// TwinCAT 3 PLC project Motion
// ProgramVersion: 3.1.4022.0
// libraries:
//   Tc2_MC2, * (Beckhoff Automation GmbH)
//   Tc2_Standard, * (Beckhoff Automation GmbH)
//   Tc2_System, * (Beckhoff Automation GmbH)
//   Tc3_Module, * (Beckhoff Automation GmbH)
//   VisuSymbols,3.5.10.0,System
// project tree:
//   / GlobalTextList.TcGTLO (not stored), PlcTask.TcTTO, VisualizationManager.TcVMO (not stored), VISU_TASK.TcTTO (not stored)
//   GVLs/ GVL_ver.TcGVL
//   POUs/ Axis2.TcPOU, Axis3.TcPOU (not stored), Axis4.TcPOU, Axis5.TcPOU (not stored), Axis6.TcPOU (not stored), Axis7.TcPOU (not stored), Axis8.TcPOU, Axis9.TcPOU (not stored), Axis10.TcPOU, GCC2.TcPOU (not stored), LadderLogic.TcPOU, MAIN.TcPOU, Axis1.TcPOU (not stored), GCC1.TcPOU
//   VISUs/ StandMotors.TcVIS, ManiMotors.TcVIS
// real-time tasks:
//   TASK PlcTask: cycle T#10ms, priority 20, ADS port 350
//   TASK VISU_TASK: cycle T#200000us, priority 30, ADS port 351
// motion (NC):
//   TASK NC-Task 1 SAF: cycle T#2ms, priority 4, ADS port 501
//   TASK NC-Task 1 SVB: cycle T#10ms, priority 8, ADS port 511
//   AXIS Axis 2 (id 2)
//     Dynamic: Acceleration=4, Deceleration=4, Jerk=4, AccelerationMaximum=4, DecelerationMaximum=4
//     Velo: RefSearch=0.3125, RefSync=0.3125, SlowManual=0.15625, FastManual=0.3125, Maximum=1
//     BacklashCompensation: Enable=true
//     OtherSettings: AllowMotionCmdToSlave=true, PulseDistancePos=0.015625, PulseDistanceNeg=0.015625
//     encoder EncType=4
//       EncPara: ScaleFactorNumerator=0.00015625, MaxCount=#x0000ffff
//         ActPosCorrection: Enable=true, Time=0.02
//         Inc: RefSoftSyncMask=#x0000ffff
//     drive DrvType=24
//       Analog: VeloReferenz=2, ScaleFactorActTorque=0.1
//       TimeComp: TaskDelayCycles=1
//     controller CtrType=1
//       CtrPara: PriorControlFactor=1
//         Observer: BandWidth=20
//   AXIS Axis 3 (id 3)
//     Dynamic: Acceleration=4, Deceleration=4, Jerk=4, AccelerationMaximum=4, DecelerationMaximum=4
//     Velo: RefSearch=0.3125, RefSync=0.3125, SlowManual=0.015625, FastManual=0.3125, Maximum=1
//     BacklashCompensation: Enable=true
//     OtherSettings: AllowMotionCmdToSlave=true, PulseDistancePos=0.015625
//     encoder EncType=4
//       EncPara: ScaleFactorNumerator=7.8125e-06, MaxCount=#x0000ffff
//         ActPosCorrection: Enable=true, Time=0.02
//         Inc: RefSoftSyncMask=#x0000ffff
//     drive DrvType=24
//       Analog: VeloReferenz=2, ScaleFactorActTorque=0.1
//       TimeComp: TaskDelayCycles=1
//     controller CtrType=1
//       CtrPara: PriorControlFactor=1
//         Observer: BandWidth=20
//   AXIS Axis 4 (id 4)
//     Dynamic: Acceleration=4, Deceleration=4, Jerk=4, AccelerationMaximum=4, DecelerationMaximum=4
//     Velo: RefSearch=0.3125, RefSync=0.3125, SlowManual=0.15625, FastManual=0.3125, Maximum=1
//     BacklashCompensation: Enable=true
//     OtherSettings: PulseDistancePos=0.015625, PulseDistanceNeg=0.015625
//     encoder EncType=4
//       EncPara: ScaleFactorNumerator=0.00015625, MaxCount=#x0000ffff
//         SoftEndMinControl: Enable=true, Range=-2.1
//         SoftEndMaxControl: Enable=true, Range=6.1
//         ActPosCorrection: Enable=true, Time=0.02
//         Inc: RefSoftSyncMask=#x0000ffff
//     drive DrvType=24
//       Analog: VeloReferenz=2, ScaleFactorActTorque=0.1
//       TimeComp: TaskDelayCycles=1
//     controller CtrType=1
//       CtrPara: PriorControlFactor=1
//         PosDiffControl: Range=1
//         Observer: BandWidth=20
//   AXIS Axis 5 (id 5)
//     Dynamic: Acceleration=4, Deceleration=4, Jerk=4, AccelerationMaximum=4, DecelerationMaximum=4
//     Velo: RefSearch=0.3125, RefSync=0.3125, SlowManual=0.15625, FastManual=0.3125, Maximum=1
//     BacklashCompensation: Enable=true
//     OtherSettings: AllowMotionCmdToSlave=true, PulseDistancePos=0.015625, PulseDistanceNeg=0.015625
//     encoder EncType=4
//       EncPara: ScaleFactorNumerator=7.8125e-06, MaxCount=#x0000ffff
//         ActPosCorrection: Enable=true, Time=0.02
//         Inc: RefSoftSyncMask=#x0000ffff
//     drive DrvType=24
//       Analog: VeloReferenz=2, ScaleFactorActTorque=0.1
//       TimeComp: TaskDelayCycles=1
//     controller CtrType=1
//       CtrPara: PriorControlFactor=1
//         Observer: BandWidth=20
//   AXIS Axis 6 (id 6)
//     Dynamic: Acceleration=4, Deceleration=4, Jerk=4, AccelerationMaximum=4, DecelerationMaximum=4
//     Velo: RefSearch=0.3125, RefSync=0.3125, SlowManual=0.15625, FastManual=0.3125, Maximum=1
//     BacklashCompensation: Enable=true
//     OtherSettings: AllowMotionCmdToSlave=true, PulseDistancePos=0.015625, PulseDistanceNeg=0.015625
//     encoder EncType=4
//       EncPara: ScaleFactorNumerator=0.00015625, MaxCount=#x0000ffff
//         ActPosCorrection: Enable=true, Time=0.02
//         Inc: RefSoftSyncMask=#x0000ffff
//     drive DrvType=24
//       Analog: VeloReferenz=2, ScaleFactorActTorque=0.1
//       TimeComp: TaskDelayCycles=1
//     controller CtrType=1
//       CtrPara: PriorControlFactor=1
//         Observer: BandWidth=20
//   AXIS Axis 7 (id 7)
//     Dynamic: Acceleration=4, Deceleration=4, Jerk=4, AccelerationMaximum=4, DecelerationMaximum=4
//     Velo: RefSearch=0.3125, RefSync=0.3125, SlowManual=0.15625, FastManual=0.3125, Maximum=1
//     BacklashCompensation: Enable=true
//     OtherSettings: AllowMotionCmdToSlave=true, PulseDistancePos=0.015625, PulseDistanceNeg=0.015625
//     encoder EncType=1
//       EncPara: ScaleFactorNumerator=1.5625e-05
//         ActPosCorrection: Enable=true, Time=0.02
//         Inc: RefSoftSyncMask=#x0000ffff
//     drive DrvType=24
//       Analog: VeloReferenz=2, ScaleFactorActTorque=0.1
//       TimeComp: TaskDelayCycles=1
//     controller CtrType=1
//       CtrPara: PriorControlFactor=1
//         Observer: BandWidth=20
//   AXIS Axis 8 (id 8)
//     Dynamic: Acceleration=4, Deceleration=4, Jerk=4, AccelerationMaximum=4, DecelerationMaximum=4
//     Velo: RefSearch=0.3125, RefSync=0.3125, SlowManual=0.15625, FastManual=0.3125, Maximum=1
//     BacklashCompensation: Enable=true
//     OtherSettings: AllowMotionCmdToSlave=true, PulseDistancePos=0.015625, PulseDistanceNeg=0.015625
//     encoder EncType=4
//       EncPara: ScaleFactorNumerator=1.5625e-05, MaxCount=#x0000ffff
//         ActPosCorrection: Enable=true, Time=0.02
//         Inc: RefSoftSyncMask=#x0000ffff
//     drive DrvType=24
//       Analog: VeloReferenz=2, ScaleFactorActTorque=0.1
//       TimeComp: TaskDelayCycles=1
//     controller CtrType=1
//       CtrPara: PriorControlFactor=1
//         Observer: BandWidth=20
//   AXIS Axis 9 (id 9)
//     Dynamic: Acceleration=4, Deceleration=4, Jerk=4, AccelerationMaximum=4, DecelerationMaximum=4
//     Velo: RefSearch=0.3125, RefSync=0.3125, SlowManual=0.15625, FastManual=0.3125, Maximum=1
//     BacklashCompensation: Enable=true
//     OtherSettings: AllowMotionCmdToSlave=true, PulseDistancePos=0.015625, PulseDistanceNeg=0.015625
//     encoder EncType=4
//       EncPara: ScaleFactorNumerator=7.812e-05, MaxCount=#x0000ffff
//         ActPosCorrection: Enable=true, Time=0.02
//         Inc: RefSoftSyncMask=#x0000ffff
//     drive DrvType=24
//       Analog: VeloReferenz=2, ScaleFactorActTorque=0.1
//       TimeComp: TaskDelayCycles=1
//     controller CtrType=1
//       CtrPara: PriorControlFactor=1
//         Observer: BandWidth=20
//   AXIS Axis 10 (id 10)
//     General: UnitName=°
//     Dynamic: Acceleration=4, Deceleration=4, Jerk=4, AccelerationMaximum=4, DecelerationMaximum=4
//     Velo: RefSearch=0.3125, RefSync=0.3125, SlowManual=0.15625, FastManual=0.3125, Maximum=1
//     BacklashCompensation: Enable=true
//     OtherSettings: AllowMotionCmdToSlave=true, PulseDistancePos=0.015625, PulseDistanceNeg=0.015625
//     encoder EncType=4
//       EncPara: ScaleFactorNumerator=0.00028125, MaxCount=#x0000ffff
//         ActPosCorrection: Enable=true, Time=0.02
//         Inc: RefSoftSyncMask=#x0000ffff
//     drive DrvType=24
//       Analog: VeloReferenz=2, ScaleFactorActTorque=0.1
//       TimeComp: TaskDelayCycles=1
//     controller CtrType=1
//       CtrPara: PriorControlFactor=1
//         Observer: BandWidth=20
//   AXIS Axis 1 (id 1)
//     Dynamic: Acceleration=4, Deceleration=4, Jerk=4, AccelerationMaximum=4, DecelerationMaximum=4
//     Velo: RefSearch=0.3125, RefSync=0.3125, SlowManual=0.15625, FastManual=0.3125, Maximum=1
//     BacklashCompensation: Enable=true
//     OtherSettings: AllowMotionCmdToSlave=true, PulseDistancePos=0.015625, PulseDistanceNeg=0.015625
//     encoder EncType=4
//       EncPara: ScaleFactorNumerator=7.8125e-06, MaxCount=#x0000ffff
//         ActPosCorrection: Enable=true, Time=0.02
//         Inc: RefMode=2, RefSoftSyncMask=#x0000ffff
//     drive DrvType=24
//       Analog: VeloReferenz=10, ScaleFactorActTorque=0.1
//       TimeComp: TaskDelayCycles=1
//     controller CtrType=1
//       CtrPara: PriorControlFactor=1
//         Observer: BandWidth=20
// I/O:
//   DEVICE Device 1 (EtherCAT), AmsNetId 5.45.61.88.2.1
//     Term 14 (EK1200) [EK1200-5000 EtherCAT Power supply (2A E-Bus)]
//       Term 15 (EL9210) [EL9210 Power Supplier with LED (24V, Fuse, Diagnostics)]
//       Term 16 (EL9576) [EL9576 Brake chopper terminal]
//       Term 17 (EL9576) [EL9576 Brake chopper terminal]
//       Term 18 (EL7047) [EL7047 1Ch. Stepper motor output stage (50V, 5A)]
//       Term 19 (EL7047) [EL7047 1Ch. Stepper motor output stage (50V, 5A)]
//       Term 20 (EL7047) [EL7047 1Ch. Stepper motor output stage (50V, 5A)]
//       Term 21 (EL7047) [EL7047 1Ch. Stepper motor output stage (50V, 5A)]
//       Term 22 (EL7047) [EL7047 1Ch. Stepper motor output stage (50V, 5A)]
//       Term 23 (EL7047) [EL7047 1Ch. Stepper motor output stage (50V, 5A)]
//       Term 24 (EL2004) [EL2004 4Ch. Dig. Output 24V, 0.5A]
//       Term 25 (EL2004) [EL2004 4Ch. Dig. Output 24V, 0.5A]
//       Term 26 (EK1110) [EK1110 EtherCAT extension]
//     Term 27 (EK1100) [EK1100 EtherCAT Coupler (2A E-Bus)]
//       Term 28 (EL9210) [EL9210 Power Supplier with LED (24V, Fuse, Diagnostics)]
//       Term 29 (EL9576) [EL9576 Brake chopper terminal]
//       Term 30 (EL7047) [EL7047 1Ch. Stepper motor output stage (50V, 5A)]
//       Term 31 (EL7047) [EL7047 1Ch. Stepper motor output stage (50V, 5A)]
//       Term 32 (EL7047) [EL7047 1Ch. Stepper motor output stage (50V, 5A)]
//       Term 33 (EL7047) [EL7047 1Ch. Stepper motor output stage (50V, 5A)]
//       Term 34 (EL5101) [EL5101 1Ch. Inc. Encoder 5V] (disabled)
//       Term 35 (EL5101) [EL5101 1Ch. Inc. Encoder 5V] (disabled)
//       Term 36 (EL5101) [EL5101 1Ch. Inc. Encoder 5V] (disabled)
//       Term 37 (EL2004) [EL2004 4Ch. Dig. Output 24V, 0.5A] (disabled)
//       Term 38 (EL9576) [EL9576 Brake chopper terminal] (disabled)
//       Term 39 (EL7047) [EL7047 1Ch. Stepper motor output stage (50V, 5A)] (disabled)
//       Term 40 (EL7047) [EL7047 1Ch. Stepper motor output stage (50V, 5A)] (disabled)
//       Term 41 (EL7031) [EL7031 1Ch. Stepper motor output stage (24V, 1.5A)] (disabled)
//       Term 42 (EL7031) [EL7031 1Ch. Stepper motor output stage (24V, 1.5A)] (disabled)
//       Term 43 (EL1104) [EL1104 4Ch. Dig. Input 24V, 3ms, Sensor Power] (disabled)
//       Term 44 (EL1104) [EL1104 4Ch. Dig. Input 24V, 3ms, Sensor Power] (disabled)
//       Term 45 (EL1104) [EL1104 4Ch. Dig. Input 24V, 3ms, Sensor Power] (disabled)
//       Term 46 (EL2004) [EL2004 4Ch. Dig. Output 24V, 0.5A] (disabled)
//       Term 47 (EL2624) [EL2624 4Ch. Relay Output, NO (125V AC / 30V DC)] (disabled)
//       Term 48 (EL9011) [EL9011 End Terminal] (disabled)
//   DEVICE Device 4 (COM Port)
// variable links:
//   NC-Task 1 SAF/Axes/Axis 1 <-> Device 1 (EtherCAT)/Term 14 (EK1200)/Term 18 (EL7047)
//     Drive/Inputs/In/nState1 @bit 3 <-> STM Status/Status/Error
//     Drive/Inputs/In/nState1 @bit 7 <-> STM Status/Status/Motor stall
//     Drive/Inputs/In/nState1 @bit 5 <-> STM Status/Status/Moving negative
//     Drive/Inputs/In/nState1 @bit 4 <-> STM Status/Status/Moving positive
//     Drive/Inputs/In/nState1 @bit 1 <-> STM Status/Status/Ready
//     Drive/Inputs/In/nState1 <-> STM Status/Status/Ready to enable
//     Drive/Inputs/In/nState1 @bit 6 <-> STM Status/Status/Torque reduced
//     Drive/Inputs/In/nState1 @bit 2 <-> STM Status/Status/Warning
//     Drive/Inputs/In/nState2 @bit 5 <-> STM Status/Status/Sync error
//     Drive/Inputs/In/nState2 @bit 7 <-> STM Status/Status/TxPDO Toggle
//     Drive/Inputs/In/nState4 @bit 1 <-> WcState/InputToggle
//     Drive/Inputs/In/nState4 <-> WcState/WcState
//     Drive/Outputs/Out/nCtrl1 <-> STM Control/Control/Enable
//     Drive/Outputs/Out/nCtrl1 @bit 2 <-> STM Control/Control/Reduce torque
//     Drive/Outputs/Out/nCtrl1 @bit 1 <-> STM Control/Control/Reset
//     Drive/Outputs/Out/nCtrl2 @bit 3 <-> STM Control/Control/Digital output 1
//     Drive/Outputs/Out/nDataOut2[0] <-> STM Velocity/Velocity
//     Enc/Inputs/In/nDataIn1[0] <-> ENC Status compact/Counter value
//     Enc/Inputs/In/nDataIn2[0] <-> ENC Status compact/Latch value
//     Enc/Inputs/In/nState1 @bit 4 <-> ENC Status compact/Status/Counter overflow
//     Enc/Inputs/In/nState1 @bit 3 <-> ENC Status compact/Status/Counter underflow
//     Enc/Inputs/In/nState1 @bit 7 <-> ENC Status compact/Status/Extrapolation stall
//     Enc/Inputs/In/nState1 <-> ENC Status compact/Status/Latch C valid
//     Enc/Inputs/In/nState1 @bit 1 <-> ENC Status compact/Status/Latch extern valid
//     Enc/Inputs/In/nState1 @bit 2 <-> ENC Status compact/Status/Set counter done
//     Enc/Inputs/In/nState2 @bit 4 <-> ENC Status compact/Status/Status of extern latch
//     Enc/Inputs/In/nState2 <-> ENC Status compact/Status/Status of input A
//     Enc/Inputs/In/nState2 @bit 1 <-> ENC Status compact/Status/Status of input B
//     Enc/Inputs/In/nState2 @bit 2 <-> ENC Status compact/Status/Status of input C
//     Enc/Inputs/In/nState2 @bit 5 <-> ENC Status compact/Status/Sync error
//     Enc/Inputs/In/nState2 @bit 7 <-> ENC Status compact/Status/TxPDO Toggle
//     Enc/Inputs/In/nState4 @bit 1 <-> WcState/InputToggle
//     Enc/Inputs/In/nState4 <-> WcState/WcState
//     Enc/Outputs/Out/nCtrl1 <-> ENC Control compact/Control/Enable latch C
//     Enc/Outputs/Out/nCtrl1 @bit 3 <-> ENC Control compact/Control/Enable latch extern on negative edge
//     Enc/Outputs/Out/nCtrl1 @bit 1 <-> ENC Control compact/Control/Enable latch extern on positive edge
//     Enc/Outputs/Out/nCtrl1 @bit 2 <-> ENC Control compact/Control/Set counter
//     Enc/Outputs/Out/nDataOut1[0] <-> ENC Control compact/Set counter value
//   NC-Task 1 SAF/Axes/Axis 10 <-> Device 1 (EtherCAT)/Term 27 (EK1100)/Term 33 (EL7047)
//     Drive/Inputs/In/nState1 @bit 3 <-> STM Status/Status/Error
//     Drive/Inputs/In/nState1 @bit 7 <-> STM Status/Status/Motor stall
//     Drive/Inputs/In/nState1 @bit 5 <-> STM Status/Status/Moving negative
//     Drive/Inputs/In/nState1 @bit 4 <-> STM Status/Status/Moving positive
//     Drive/Inputs/In/nState1 @bit 1 <-> STM Status/Status/Ready
//     Drive/Inputs/In/nState1 <-> STM Status/Status/Ready to enable
//     Drive/Inputs/In/nState1 @bit 6 <-> STM Status/Status/Torque reduced
//     Drive/Inputs/In/nState1 @bit 2 <-> STM Status/Status/Warning
//     Drive/Inputs/In/nState2 @bit 3 <-> STM Status/Status/Digital input 1
//     Drive/Inputs/In/nState2 @bit 4 <-> STM Status/Status/Digital input 2
//     Drive/Inputs/In/nState2 @bit 5 <-> STM Status/Status/Sync error
//     Drive/Inputs/In/nState2 @bit 7 <-> STM Status/Status/TxPDO Toggle
//     Drive/Inputs/In/nState4 @bit 1 <-> WcState/InputToggle
//     Drive/Inputs/In/nState4 <-> WcState/WcState
//     Drive/Outputs/Out/nCtrl1 <-> STM Control/Control/Enable
//     Drive/Outputs/Out/nCtrl1 @bit 2 <-> STM Control/Control/Reduce torque
//     Drive/Outputs/Out/nCtrl1 @bit 1 <-> STM Control/Control/Reset
//     Drive/Outputs/Out/nCtrl2 @bit 3 <-> STM Control/Control/Digital output 1
//     Drive/Outputs/Out/nDataOut2[0] <-> STM Velocity/Velocity
//     Enc/Inputs/In/nDataIn1[0] <-> ENC Status compact/Counter value
//     Enc/Inputs/In/nDataIn2[0] <-> ENC Status compact/Latch value
//     Enc/Inputs/In/nState1 @bit 4 <-> ENC Status compact/Status/Counter overflow
//     Enc/Inputs/In/nState1 @bit 3 <-> ENC Status compact/Status/Counter underflow
//     Enc/Inputs/In/nState1 @bit 7 <-> ENC Status compact/Status/Extrapolation stall
//     Enc/Inputs/In/nState1 <-> ENC Status compact/Status/Latch C valid
//     Enc/Inputs/In/nState1 @bit 1 <-> ENC Status compact/Status/Latch extern valid
//     Enc/Inputs/In/nState1 @bit 2 <-> ENC Status compact/Status/Set counter done
//     Enc/Inputs/In/nState2 @bit 4 <-> ENC Status compact/Status/Status of extern latch
//     Enc/Inputs/In/nState2 <-> ENC Status compact/Status/Status of input A
//     Enc/Inputs/In/nState2 @bit 1 <-> ENC Status compact/Status/Status of input B
//     Enc/Inputs/In/nState2 @bit 2 <-> ENC Status compact/Status/Status of input C
//     Enc/Inputs/In/nState2 @bit 5 <-> ENC Status compact/Status/Sync error
//     Enc/Inputs/In/nState2 @bit 7 <-> ENC Status compact/Status/TxPDO Toggle
//     Enc/Inputs/In/nState4 @bit 1 <-> WcState/InputToggle
//     Enc/Inputs/In/nState4 <-> WcState/WcState
//     Enc/Outputs/Out/nCtrl1 <-> ENC Control compact/Control/Enable latch C
//     Enc/Outputs/Out/nCtrl1 @bit 3 <-> ENC Control compact/Control/Enable latch extern on negative edge
//     Enc/Outputs/Out/nCtrl1 @bit 1 <-> ENC Control compact/Control/Enable latch extern on positive edge
//     Enc/Outputs/Out/nCtrl1 @bit 2 <-> ENC Control compact/Control/Set counter
//     Enc/Outputs/Out/nDataOut1[0] <-> ENC Control compact/Set counter value
//   NC-Task 1 SAF/Axes/Axis 2 <-> Device 1 (EtherCAT)/Term 14 (EK1200)/Term 19 (EL7047)
//     Drive/Inputs/In/nState1 @bit 3 <-> STM Status/Status/Error
//     Drive/Inputs/In/nState1 @bit 7 <-> STM Status/Status/Motor stall
//     Drive/Inputs/In/nState1 @bit 5 <-> STM Status/Status/Moving negative
//     Drive/Inputs/In/nState1 @bit 4 <-> STM Status/Status/Moving positive
//     Drive/Inputs/In/nState1 @bit 1 <-> STM Status/Status/Ready
//     Drive/Inputs/In/nState1 <-> STM Status/Status/Ready to enable
//     Drive/Inputs/In/nState1 @bit 6 <-> STM Status/Status/Torque reduced
//     Drive/Inputs/In/nState1 @bit 2 <-> STM Status/Status/Warning
//     Drive/Inputs/In/nState2 @bit 5 <-> STM Status/Status/Sync error
//     Drive/Inputs/In/nState2 @bit 7 <-> STM Status/Status/TxPDO Toggle
//     Drive/Inputs/In/nState4 @bit 1 <-> WcState/InputToggle
//     Drive/Inputs/In/nState4 <-> WcState/WcState
//     Drive/Outputs/Out/nCtrl1 <-> STM Control/Control/Enable
//     Drive/Outputs/Out/nCtrl1 @bit 2 <-> STM Control/Control/Reduce torque
//     Drive/Outputs/Out/nCtrl1 @bit 1 <-> STM Control/Control/Reset
//     Drive/Outputs/Out/nCtrl2 @bit 3 <-> STM Control/Control/Digital output 1
//     Drive/Outputs/Out/nDataOut2[0] <-> STM Velocity/Velocity
//     Enc/Inputs/In/nDataIn1[0] <-> ENC Status compact/Counter value
//     Enc/Inputs/In/nDataIn2[0] <-> ENC Status compact/Latch value
//     Enc/Inputs/In/nState1 @bit 4 <-> ENC Status compact/Status/Counter overflow
//     Enc/Inputs/In/nState1 @bit 3 <-> ENC Status compact/Status/Counter underflow
//     Enc/Inputs/In/nState1 @bit 7 <-> ENC Status compact/Status/Extrapolation stall
//     Enc/Inputs/In/nState1 <-> ENC Status compact/Status/Latch C valid
//     Enc/Inputs/In/nState1 @bit 1 <-> ENC Status compact/Status/Latch extern valid
//     Enc/Inputs/In/nState1 @bit 2 <-> ENC Status compact/Status/Set counter done
//     Enc/Inputs/In/nState2 @bit 4 <-> ENC Status compact/Status/Status of extern latch
//     Enc/Inputs/In/nState2 <-> ENC Status compact/Status/Status of input A
//     Enc/Inputs/In/nState2 @bit 1 <-> ENC Status compact/Status/Status of input B
//     Enc/Inputs/In/nState2 @bit 2 <-> ENC Status compact/Status/Status of input C
//     Enc/Inputs/In/nState2 @bit 5 <-> ENC Status compact/Status/Sync error
//     Enc/Inputs/In/nState2 @bit 7 <-> ENC Status compact/Status/TxPDO Toggle
//     Enc/Inputs/In/nState4 @bit 1 <-> WcState/InputToggle
//     Enc/Inputs/In/nState4 <-> WcState/WcState
//     Enc/Outputs/Out/nCtrl1 <-> ENC Control compact/Control/Enable latch C
//     Enc/Outputs/Out/nCtrl1 @bit 3 <-> ENC Control compact/Control/Enable latch extern on negative edge
//     Enc/Outputs/Out/nCtrl1 @bit 1 <-> ENC Control compact/Control/Enable latch extern on positive edge
//     Enc/Outputs/Out/nCtrl1 @bit 2 <-> ENC Control compact/Control/Set counter
//     Enc/Outputs/Out/nDataOut1[0] <-> ENC Control compact/Set counter value
//   NC-Task 1 SAF/Axes/Axis 3 <-> Device 1 (EtherCAT)/Term 14 (EK1200)/Term 20 (EL7047)
//     Drive/Inputs/In/nState1 @bit 3 <-> STM Status/Status/Error
//     Drive/Inputs/In/nState1 @bit 7 <-> STM Status/Status/Motor stall
//     Drive/Inputs/In/nState1 @bit 5 <-> STM Status/Status/Moving negative
//     Drive/Inputs/In/nState1 @bit 4 <-> STM Status/Status/Moving positive
//     Drive/Inputs/In/nState1 @bit 1 <-> STM Status/Status/Ready
//     Drive/Inputs/In/nState1 <-> STM Status/Status/Ready to enable
//     Drive/Inputs/In/nState1 @bit 6 <-> STM Status/Status/Torque reduced
//     Drive/Inputs/In/nState1 @bit 2 <-> STM Status/Status/Warning
//     Drive/Inputs/In/nState2 @bit 5 <-> STM Status/Status/Sync error
//     Drive/Inputs/In/nState2 @bit 7 <-> STM Status/Status/TxPDO Toggle
//     Drive/Inputs/In/nState4 @bit 1 <-> WcState/InputToggle
//     Drive/Inputs/In/nState4 <-> WcState/WcState
//     Drive/Outputs/Out/nCtrl1 <-> STM Control/Control/Enable
//     Drive/Outputs/Out/nCtrl1 @bit 2 <-> STM Control/Control/Reduce torque
//     Drive/Outputs/Out/nCtrl1 @bit 1 <-> STM Control/Control/Reset
//     Drive/Outputs/Out/nCtrl2 @bit 3 <-> STM Control/Control/Digital output 1
//     Drive/Outputs/Out/nDataOut2[0] <-> STM Velocity/Velocity
//     Enc/Inputs/In/nDataIn1[0] <-> ENC Status compact/Counter value
//     Enc/Inputs/In/nDataIn2[0] <-> ENC Status compact/Latch value
//     Enc/Inputs/In/nState1 @bit 4 <-> ENC Status compact/Status/Counter overflow
//     Enc/Inputs/In/nState1 @bit 3 <-> ENC Status compact/Status/Counter underflow
//     Enc/Inputs/In/nState1 @bit 7 <-> ENC Status compact/Status/Extrapolation stall
//     Enc/Inputs/In/nState1 <-> ENC Status compact/Status/Latch C valid
//     Enc/Inputs/In/nState1 @bit 1 <-> ENC Status compact/Status/Latch extern valid
//     Enc/Inputs/In/nState1 @bit 2 <-> ENC Status compact/Status/Set counter done
//     Enc/Inputs/In/nState2 @bit 4 <-> ENC Status compact/Status/Status of extern latch
//     Enc/Inputs/In/nState2 <-> ENC Status compact/Status/Status of input A
//     Enc/Inputs/In/nState2 @bit 1 <-> ENC Status compact/Status/Status of input B
//     Enc/Inputs/In/nState2 @bit 2 <-> ENC Status compact/Status/Status of input C
//     Enc/Inputs/In/nState2 @bit 5 <-> ENC Status compact/Status/Sync error
//     Enc/Inputs/In/nState2 @bit 7 <-> ENC Status compact/Status/TxPDO Toggle
//     Enc/Inputs/In/nState4 @bit 1 <-> WcState/InputToggle
//     Enc/Inputs/In/nState4 <-> WcState/WcState
//     Enc/Outputs/Out/nCtrl1 <-> ENC Control compact/Control/Enable latch C
//     Enc/Outputs/Out/nCtrl1 @bit 3 <-> ENC Control compact/Control/Enable latch extern on negative edge
//     Enc/Outputs/Out/nCtrl1 @bit 1 <-> ENC Control compact/Control/Enable latch extern on positive edge
//     Enc/Outputs/Out/nCtrl1 @bit 2 <-> ENC Control compact/Control/Set counter
//     Enc/Outputs/Out/nDataOut1[0] <-> ENC Control compact/Set counter value
//   NC-Task 1 SAF/Axes/Axis 4 <-> Device 1 (EtherCAT)/Term 14 (EK1200)/Term 21 (EL7047)
//     Drive/Inputs/In/nState1 @bit 3 <-> STM Status/Status/Error
//     Drive/Inputs/In/nState1 @bit 7 <-> STM Status/Status/Motor stall
//     Drive/Inputs/In/nState1 @bit 5 <-> STM Status/Status/Moving negative
//     Drive/Inputs/In/nState1 @bit 4 <-> STM Status/Status/Moving positive
//     Drive/Inputs/In/nState1 @bit 1 <-> STM Status/Status/Ready
//     Drive/Inputs/In/nState1 <-> STM Status/Status/Ready to enable
//     Drive/Inputs/In/nState1 @bit 6 <-> STM Status/Status/Torque reduced
//     Drive/Inputs/In/nState1 @bit 2 <-> STM Status/Status/Warning
//     Drive/Inputs/In/nState2 @bit 5 <-> STM Status/Status/Sync error
//     Drive/Inputs/In/nState2 @bit 7 <-> STM Status/Status/TxPDO Toggle
//     Drive/Inputs/In/nState4 @bit 1 <-> WcState/InputToggle
//     Drive/Inputs/In/nState4 <-> WcState/WcState
//     Drive/Outputs/Out/nCtrl1 <-> STM Control/Control/Enable
//     Drive/Outputs/Out/nCtrl1 @bit 2 <-> STM Control/Control/Reduce torque
//     Drive/Outputs/Out/nCtrl1 @bit 1 <-> STM Control/Control/Reset
//     Drive/Outputs/Out/nCtrl2 @bit 3 <-> STM Control/Control/Digital output 1
//     Drive/Outputs/Out/nDataOut2[0] <-> STM Velocity/Velocity
//     Enc/Inputs/In/nDataIn1[0] <-> ENC Status compact/Counter value
//     Enc/Inputs/In/nDataIn2[0] <-> ENC Status compact/Latch value
//     Enc/Inputs/In/nState1 @bit 4 <-> ENC Status compact/Status/Counter overflow
//     Enc/Inputs/In/nState1 @bit 3 <-> ENC Status compact/Status/Counter underflow
//     Enc/Inputs/In/nState1 @bit 7 <-> ENC Status compact/Status/Extrapolation stall
//     Enc/Inputs/In/nState1 <-> ENC Status compact/Status/Latch C valid
//     Enc/Inputs/In/nState1 @bit 1 <-> ENC Status compact/Status/Latch extern valid
//     Enc/Inputs/In/nState1 @bit 2 <-> ENC Status compact/Status/Set counter done
//     Enc/Inputs/In/nState2 @bit 4 <-> ENC Status compact/Status/Status of extern latch
//     Enc/Inputs/In/nState2 <-> ENC Status compact/Status/Status of input A
//     Enc/Inputs/In/nState2 @bit 1 <-> ENC Status compact/Status/Status of input B
//     Enc/Inputs/In/nState2 @bit 2 <-> ENC Status compact/Status/Status of input C
//     Enc/Inputs/In/nState2 @bit 5 <-> ENC Status compact/Status/Sync error
//     Enc/Inputs/In/nState2 @bit 7 <-> ENC Status compact/Status/TxPDO Toggle
//     Enc/Inputs/In/nState4 @bit 1 <-> WcState/InputToggle
//     Enc/Inputs/In/nState4 <-> WcState/WcState
//     Enc/Outputs/Out/nCtrl1 <-> ENC Control compact/Control/Enable latch C
//     Enc/Outputs/Out/nCtrl1 @bit 3 <-> ENC Control compact/Control/Enable latch extern on negative edge
//     Enc/Outputs/Out/nCtrl1 @bit 1 <-> ENC Control compact/Control/Enable latch extern on positive edge
//     Enc/Outputs/Out/nCtrl1 @bit 2 <-> ENC Control compact/Control/Set counter
//     Enc/Outputs/Out/nDataOut1[0] <-> ENC Control compact/Set counter value
//   NC-Task 1 SAF/Axes/Axis 5 <-> Device 1 (EtherCAT)/Term 14 (EK1200)/Term 22 (EL7047)
//     Drive/Inputs/In/nState1 @bit 3 <-> STM Status/Status/Error
//     Drive/Inputs/In/nState1 @bit 7 <-> STM Status/Status/Motor stall
//     Drive/Inputs/In/nState1 @bit 5 <-> STM Status/Status/Moving negative
//     Drive/Inputs/In/nState1 @bit 4 <-> STM Status/Status/Moving positive
//     Drive/Inputs/In/nState1 @bit 1 <-> STM Status/Status/Ready
//     Drive/Inputs/In/nState1 <-> STM Status/Status/Ready to enable
//     Drive/Inputs/In/nState1 @bit 6 <-> STM Status/Status/Torque reduced
//     Drive/Inputs/In/nState1 @bit 2 <-> STM Status/Status/Warning
//     Drive/Inputs/In/nState2 @bit 5 <-> STM Status/Status/Sync error
//     Drive/Inputs/In/nState2 @bit 7 <-> STM Status/Status/TxPDO Toggle
//     Drive/Inputs/In/nState4 @bit 1 <-> WcState/InputToggle
//     Drive/Inputs/In/nState4 <-> WcState/WcState
//     Drive/Outputs/Out/nCtrl1 <-> STM Control/Control/Enable
//     Drive/Outputs/Out/nCtrl1 @bit 2 <-> STM Control/Control/Reduce torque
//     Drive/Outputs/Out/nCtrl1 @bit 1 <-> STM Control/Control/Reset
//     Drive/Outputs/Out/nCtrl2 @bit 3 <-> STM Control/Control/Digital output 1
//     Drive/Outputs/Out/nDataOut2[0] <-> STM Velocity/Velocity
//     Enc/Inputs/In/nDataIn1[0] <-> ENC Status compact/Counter value
//     Enc/Inputs/In/nDataIn2[0] <-> ENC Status compact/Latch value
//     Enc/Inputs/In/nState1 @bit 4 <-> ENC Status compact/Status/Counter overflow
//     Enc/Inputs/In/nState1 @bit 3 <-> ENC Status compact/Status/Counter underflow
//     Enc/Inputs/In/nState1 @bit 7 <-> ENC Status compact/Status/Extrapolation stall
//     Enc/Inputs/In/nState1 <-> ENC Status compact/Status/Latch C valid
//     Enc/Inputs/In/nState1 @bit 1 <-> ENC Status compact/Status/Latch extern valid
//     Enc/Inputs/In/nState1 @bit 2 <-> ENC Status compact/Status/Set counter done
//     Enc/Inputs/In/nState2 @bit 4 <-> ENC Status compact/Status/Status of extern latch
//     Enc/Inputs/In/nState2 <-> ENC Status compact/Status/Status of input A
//     Enc/Inputs/In/nState2 @bit 1 <-> ENC Status compact/Status/Status of input B
//     Enc/Inputs/In/nState2 @bit 2 <-> ENC Status compact/Status/Status of input C
//     Enc/Inputs/In/nState2 @bit 5 <-> ENC Status compact/Status/Sync error
//     Enc/Inputs/In/nState2 @bit 7 <-> ENC Status compact/Status/TxPDO Toggle
//     Enc/Inputs/In/nState4 @bit 1 <-> WcState/InputToggle
//     Enc/Inputs/In/nState4 <-> WcState/WcState
//     Enc/Outputs/Out/nCtrl1 <-> ENC Control compact/Control/Enable latch C
//     Enc/Outputs/Out/nCtrl1 @bit 3 <-> ENC Control compact/Control/Enable latch extern on negative edge
//     Enc/Outputs/Out/nCtrl1 @bit 1 <-> ENC Control compact/Control/Enable latch extern on positive edge
//     Enc/Outputs/Out/nCtrl1 @bit 2 <-> ENC Control compact/Control/Set counter
//     Enc/Outputs/Out/nDataOut1[0] <-> ENC Control compact/Set counter value
//   NC-Task 1 SAF/Axes/Axis 6 <-> Device 1 (EtherCAT)/Term 14 (EK1200)/Term 23 (EL7047)
//     Drive/Inputs/In/nState1 @bit 3 <-> STM Status/Status/Error
//     Drive/Inputs/In/nState1 @bit 7 <-> STM Status/Status/Motor stall
//     Drive/Inputs/In/nState1 @bit 5 <-> STM Status/Status/Moving negative
//     Drive/Inputs/In/nState1 @bit 4 <-> STM Status/Status/Moving positive
//     Drive/Inputs/In/nState1 @bit 1 <-> STM Status/Status/Ready
//     Drive/Inputs/In/nState1 <-> STM Status/Status/Ready to enable
//     Drive/Inputs/In/nState1 @bit 6 <-> STM Status/Status/Torque reduced
//     Drive/Inputs/In/nState1 @bit 2 <-> STM Status/Status/Warning
//     Drive/Inputs/In/nState2 @bit 5 <-> STM Status/Status/Sync error
//     Drive/Inputs/In/nState2 @bit 7 <-> STM Status/Status/TxPDO Toggle
//     Drive/Inputs/In/nState4 @bit 1 <-> WcState/InputToggle
//     Drive/Inputs/In/nState4 <-> WcState/WcState
//     Drive/Outputs/Out/nCtrl1 <-> STM Control/Control/Enable
//     Drive/Outputs/Out/nCtrl1 @bit 2 <-> STM Control/Control/Reduce torque
//     Drive/Outputs/Out/nCtrl1 @bit 1 <-> STM Control/Control/Reset
//     Drive/Outputs/Out/nCtrl2 @bit 3 <-> STM Control/Control/Digital output 1
//     Drive/Outputs/Out/nDataOut2[0] <-> STM Velocity/Velocity
//     Enc/Inputs/In/nDataIn1[0] <-> ENC Status compact/Counter value
//     Enc/Inputs/In/nDataIn2[0] <-> ENC Status compact/Latch value
//     Enc/Inputs/In/nState1 @bit 4 <-> ENC Status compact/Status/Counter overflow
//     Enc/Inputs/In/nState1 @bit 3 <-> ENC Status compact/Status/Counter underflow
//     Enc/Inputs/In/nState1 @bit 7 <-> ENC Status compact/Status/Extrapolation stall
//     Enc/Inputs/In/nState1 <-> ENC Status compact/Status/Latch C valid
//     Enc/Inputs/In/nState1 @bit 1 <-> ENC Status compact/Status/Latch extern valid
//     Enc/Inputs/In/nState1 @bit 2 <-> ENC Status compact/Status/Set counter done
//     Enc/Inputs/In/nState2 @bit 4 <-> ENC Status compact/Status/Status of extern latch
//     Enc/Inputs/In/nState2 <-> ENC Status compact/Status/Status of input A
//     Enc/Inputs/In/nState2 @bit 1 <-> ENC Status compact/Status/Status of input B
//     Enc/Inputs/In/nState2 @bit 2 <-> ENC Status compact/Status/Status of input C
//     Enc/Inputs/In/nState2 @bit 5 <-> ENC Status compact/Status/Sync error
//     Enc/Inputs/In/nState2 @bit 7 <-> ENC Status compact/Status/TxPDO Toggle
//     Enc/Inputs/In/nState4 @bit 1 <-> WcState/InputToggle
//     Enc/Inputs/In/nState4 <-> WcState/WcState
//     Enc/Outputs/Out/nCtrl1 <-> ENC Control compact/Control/Enable latch C
//     Enc/Outputs/Out/nCtrl1 @bit 3 <-> ENC Control compact/Control/Enable latch extern on negative edge
//     Enc/Outputs/Out/nCtrl1 @bit 1 <-> ENC Control compact/Control/Enable latch extern on positive edge
//     Enc/Outputs/Out/nCtrl1 @bit 2 <-> ENC Control compact/Control/Set counter
//     Enc/Outputs/Out/nDataOut1[0] <-> ENC Control compact/Set counter value
//   NC-Task 1 SAF/Axes/Axis 7 <-> Device 1 (EtherCAT)/Term 27 (EK1100)/Term 30 (EL7047)
//     Drive/Inputs/In/nState1 @bit 3 <-> STM Status/Status/Error
//     Drive/Inputs/In/nState1 @bit 7 <-> STM Status/Status/Motor stall
//     Drive/Inputs/In/nState1 @bit 5 <-> STM Status/Status/Moving negative
//     Drive/Inputs/In/nState1 @bit 4 <-> STM Status/Status/Moving positive
//     Drive/Inputs/In/nState1 @bit 1 <-> STM Status/Status/Ready
//     Drive/Inputs/In/nState1 <-> STM Status/Status/Ready to enable
//     Drive/Inputs/In/nState1 @bit 6 <-> STM Status/Status/Torque reduced
//     Drive/Inputs/In/nState1 @bit 2 <-> STM Status/Status/Warning
//     Drive/Inputs/In/nState2 @bit 5 <-> STM Status/Status/Sync error
//     Drive/Inputs/In/nState2 @bit 7 <-> STM Status/Status/TxPDO Toggle
//     Drive/Inputs/In/nState4 @bit 1 <-> WcState/InputToggle
//     Drive/Inputs/In/nState4 <-> WcState/WcState
//     Drive/Outputs/Out/nCtrl1 <-> STM Control/Control/Enable
//     Drive/Outputs/Out/nCtrl1 @bit 2 <-> STM Control/Control/Reduce torque
//     Drive/Outputs/Out/nCtrl1 @bit 1 <-> STM Control/Control/Reset
//     Drive/Outputs/Out/nCtrl2 @bit 3 <-> STM Control/Control/Digital output 1
//     Drive/Outputs/Out/nDataOut2[0] <-> STM Velocity/Velocity
//     Enc/Inputs/In/nDataIn1[0] <-> ENC Status compact/Counter value
//     Enc/Inputs/In/nDataIn2[0] <-> ENC Status compact/Latch value
//     Enc/Inputs/In/nState1 @bit 4 <-> ENC Status compact/Status/Counter overflow
//     Enc/Inputs/In/nState1 @bit 3 <-> ENC Status compact/Status/Counter underflow
//     Enc/Inputs/In/nState1 @bit 7 <-> ENC Status compact/Status/Extrapolation stall
//     Enc/Inputs/In/nState1 <-> ENC Status compact/Status/Latch C valid
//     Enc/Inputs/In/nState1 @bit 1 <-> ENC Status compact/Status/Latch extern valid
//     Enc/Inputs/In/nState1 @bit 2 <-> ENC Status compact/Status/Set counter done
//     Enc/Inputs/In/nState2 @bit 4 <-> ENC Status compact/Status/Status of extern latch
//     Enc/Inputs/In/nState2 <-> ENC Status compact/Status/Status of input A
//     Enc/Inputs/In/nState2 @bit 1 <-> ENC Status compact/Status/Status of input B
//     Enc/Inputs/In/nState2 @bit 2 <-> ENC Status compact/Status/Status of input C
//     Enc/Inputs/In/nState2 @bit 5 <-> ENC Status compact/Status/Sync error
//     Enc/Inputs/In/nState2 @bit 7 <-> ENC Status compact/Status/TxPDO Toggle
//     Enc/Inputs/In/nState4 @bit 1 <-> WcState/InputToggle
//     Enc/Inputs/In/nState4 <-> WcState/WcState
//     Enc/Outputs/Out/nCtrl1 <-> ENC Control compact/Control/Enable latch C
//     Enc/Outputs/Out/nCtrl1 @bit 3 <-> ENC Control compact/Control/Enable latch extern on negative edge
//     Enc/Outputs/Out/nCtrl1 @bit 1 <-> ENC Control compact/Control/Enable latch extern on positive edge
//     Enc/Outputs/Out/nCtrl1 @bit 2 <-> ENC Control compact/Control/Set counter
//     Enc/Outputs/Out/nDataOut1[0] <-> ENC Control compact/Set counter value
//   NC-Task 1 SAF/Axes/Axis 8 <-> Device 1 (EtherCAT)/Term 27 (EK1100)/Term 31 (EL7047)
//     Drive/Inputs/In/nState1 @bit 3 <-> STM Status/Status/Error
//     Drive/Inputs/In/nState1 @bit 7 <-> STM Status/Status/Motor stall
//     Drive/Inputs/In/nState1 @bit 5 <-> STM Status/Status/Moving negative
//     Drive/Inputs/In/nState1 @bit 4 <-> STM Status/Status/Moving positive
//     Drive/Inputs/In/nState1 @bit 1 <-> STM Status/Status/Ready
//     Drive/Inputs/In/nState1 <-> STM Status/Status/Ready to enable
//     Drive/Inputs/In/nState1 @bit 6 <-> STM Status/Status/Torque reduced
//     Drive/Inputs/In/nState1 @bit 2 <-> STM Status/Status/Warning
//     Drive/Inputs/In/nState2 @bit 3 <-> STM Status/Status/Digital input 1
//     Drive/Inputs/In/nState2 @bit 4 <-> STM Status/Status/Digital input 2
//     Drive/Inputs/In/nState2 @bit 5 <-> STM Status/Status/Sync error
//     Drive/Inputs/In/nState2 @bit 7 <-> STM Status/Status/TxPDO Toggle
//     Drive/Inputs/In/nState4 @bit 1 <-> WcState/InputToggle
//     Drive/Inputs/In/nState4 <-> WcState/WcState
//     Drive/Outputs/Out/nCtrl1 <-> STM Control/Control/Enable
//     Drive/Outputs/Out/nCtrl1 @bit 2 <-> STM Control/Control/Reduce torque
//     Drive/Outputs/Out/nCtrl1 @bit 1 <-> STM Control/Control/Reset
//     Drive/Outputs/Out/nCtrl2 @bit 3 <-> STM Control/Control/Digital output 1
//     Drive/Outputs/Out/nDataOut2[0] <-> STM Velocity/Velocity
//     Enc/Inputs/In/nDataIn1[0] <-> ENC Status compact/Counter value
//     Enc/Inputs/In/nDataIn2[0] <-> ENC Status compact/Latch value
//     Enc/Inputs/In/nState1 @bit 4 <-> ENC Status compact/Status/Counter overflow
//     Enc/Inputs/In/nState1 @bit 3 <-> ENC Status compact/Status/Counter underflow
//     Enc/Inputs/In/nState1 @bit 7 <-> ENC Status compact/Status/Extrapolation stall
//     Enc/Inputs/In/nState1 <-> ENC Status compact/Status/Latch C valid
//     Enc/Inputs/In/nState1 @bit 1 <-> ENC Status compact/Status/Latch extern valid
//     Enc/Inputs/In/nState1 @bit 2 <-> ENC Status compact/Status/Set counter done
//     Enc/Inputs/In/nState2 @bit 4 <-> ENC Status compact/Status/Status of extern latch
//     Enc/Inputs/In/nState2 <-> ENC Status compact/Status/Status of input A
//     Enc/Inputs/In/nState2 @bit 1 <-> ENC Status compact/Status/Status of input B
//     Enc/Inputs/In/nState2 @bit 2 <-> ENC Status compact/Status/Status of input C
//     Enc/Inputs/In/nState2 @bit 5 <-> ENC Status compact/Status/Sync error
//     Enc/Inputs/In/nState2 @bit 7 <-> ENC Status compact/Status/TxPDO Toggle
//     Enc/Inputs/In/nState4 @bit 1 <-> WcState/InputToggle
//     Enc/Inputs/In/nState4 <-> WcState/WcState
//     Enc/Outputs/Out/nCtrl1 <-> ENC Control compact/Control/Enable latch C
//     Enc/Outputs/Out/nCtrl1 @bit 3 <-> ENC Control compact/Control/Enable latch extern on negative edge
//     Enc/Outputs/Out/nCtrl1 @bit 1 <-> ENC Control compact/Control/Enable latch extern on positive edge
//     Enc/Outputs/Out/nCtrl1 @bit 2 <-> ENC Control compact/Control/Set counter
//     Enc/Outputs/Out/nDataOut1[0] <-> ENC Control compact/Set counter value
//   NC-Task 1 SAF/Axes/Axis 9 <-> Device 1 (EtherCAT)/Term 27 (EK1100)/Term 32 (EL7047)
//     Drive/Inputs/In/nState1 @bit 3 <-> STM Status/Status/Error
//     Drive/Inputs/In/nState1 @bit 7 <-> STM Status/Status/Motor stall
//     Drive/Inputs/In/nState1 @bit 5 <-> STM Status/Status/Moving negative
//     Drive/Inputs/In/nState1 @bit 4 <-> STM Status/Status/Moving positive
//     Drive/Inputs/In/nState1 @bit 1 <-> STM Status/Status/Ready
//     Drive/Inputs/In/nState1 <-> STM Status/Status/Ready to enable
//     Drive/Inputs/In/nState1 @bit 6 <-> STM Status/Status/Torque reduced
//     Drive/Inputs/In/nState1 @bit 2 <-> STM Status/Status/Warning
//     Drive/Inputs/In/nState2 @bit 3 <-> STM Status/Status/Digital input 1
//     Drive/Inputs/In/nState2 @bit 4 <-> STM Status/Status/Digital input 2
//     Drive/Inputs/In/nState2 @bit 5 <-> STM Status/Status/Sync error
//     Drive/Inputs/In/nState2 @bit 7 <-> STM Status/Status/TxPDO Toggle
//     Drive/Inputs/In/nState4 @bit 1 <-> WcState/InputToggle
//     Drive/Inputs/In/nState4 <-> WcState/WcState
//     Drive/Outputs/Out/nCtrl1 <-> STM Control/Control/Enable
//     Drive/Outputs/Out/nCtrl1 @bit 2 <-> STM Control/Control/Reduce torque
//     Drive/Outputs/Out/nCtrl1 @bit 1 <-> STM Control/Control/Reset
//     Drive/Outputs/Out/nCtrl2 @bit 3 <-> STM Control/Control/Digital output 1
//     Drive/Outputs/Out/nDataOut2[0] <-> STM Velocity/Velocity
//     Enc/Inputs/In/nDataIn1[0] <-> ENC Status compact/Counter value
//     Enc/Inputs/In/nDataIn2[0] <-> ENC Status compact/Latch value
//     Enc/Inputs/In/nState1 @bit 4 <-> ENC Status compact/Status/Counter overflow
//     Enc/Inputs/In/nState1 @bit 3 <-> ENC Status compact/Status/Counter underflow
//     Enc/Inputs/In/nState1 @bit 7 <-> ENC Status compact/Status/Extrapolation stall
//     Enc/Inputs/In/nState1 <-> ENC Status compact/Status/Latch C valid
//     Enc/Inputs/In/nState1 @bit 1 <-> ENC Status compact/Status/Latch extern valid
//     Enc/Inputs/In/nState1 @bit 2 <-> ENC Status compact/Status/Set counter done
//     Enc/Inputs/In/nState2 @bit 4 <-> ENC Status compact/Status/Status of extern latch
//     Enc/Inputs/In/nState2 <-> ENC Status compact/Status/Status of input A
//     Enc/Inputs/In/nState2 @bit 1 <-> ENC Status compact/Status/Status of input B
//     Enc/Inputs/In/nState2 @bit 2 <-> ENC Status compact/Status/Status of input C
//     Enc/Inputs/In/nState2 @bit 5 <-> ENC Status compact/Status/Sync error
//     Enc/Inputs/In/nState2 @bit 7 <-> ENC Status compact/Status/TxPDO Toggle
//     Enc/Inputs/In/nState4 @bit 1 <-> WcState/InputToggle
//     Enc/Inputs/In/nState4 <-> WcState/WcState
//     Enc/Outputs/Out/nCtrl1 <-> ENC Control compact/Control/Enable latch C
//     Enc/Outputs/Out/nCtrl1 @bit 3 <-> ENC Control compact/Control/Enable latch extern on negative edge
//     Enc/Outputs/Out/nCtrl1 @bit 1 <-> ENC Control compact/Control/Enable latch extern on positive edge
//     Enc/Outputs/Out/nCtrl1 @bit 2 <-> ENC Control compact/Control/Set counter
//     Enc/Outputs/Out/nDataOut1[0] <-> ENC Control compact/Set counter value
//   Motion/Motion Instance <-> Device 1 (EtherCAT)/Term 14 (EK1200)/Term 18 (EL7047)
//     PlcTask Inputs/Axis1.biLimBwd <-> STM Status/Status/Digital input 2
//     PlcTask Inputs/Axis1.biLimFwd <-> STM Status/Status/Digital input 1
//   Motion/Motion Instance <-> Device 1 (EtherCAT)/Term 14 (EK1200)/Term 19 (EL7047)
//     PlcTask Inputs/Axis2.biLimBwd <-> STM Status/Status/Digital input 2
//     PlcTask Inputs/Axis2.biLimFwd <-> STM Status/Status/Digital input 1
//   Motion/Motion Instance <-> Device 1 (EtherCAT)/Term 14 (EK1200)/Term 20 (EL7047)
//     PlcTask Inputs/Axis3.biLimBwd <-> STM Status/Status/Digital input 2
//     PlcTask Inputs/Axis3.biLimFwd <-> STM Status/Status/Digital input 1
//   Motion/Motion Instance <-> Device 1 (EtherCAT)/Term 14 (EK1200)/Term 21 (EL7047)
//     PlcTask Inputs/Axis4.biLimBwd <-> STM Status/Status/Digital input 2
//     PlcTask Inputs/Axis4.biLimFwd <-> STM Status/Status/Digital input 1
//   Motion/Motion Instance <-> Device 1 (EtherCAT)/Term 14 (EK1200)/Term 22 (EL7047)
//     PlcTask Inputs/Axis5.biLimBwd <-> STM Status/Status/Digital input 2
//     PlcTask Inputs/Axis5.biLimFwd <-> STM Status/Status/Digital input 1
//   Motion/Motion Instance <-> Device 1 (EtherCAT)/Term 14 (EK1200)/Term 23 (EL7047)
//     PlcTask Inputs/Axis6.biLimBwd <-> STM Status/Status/Digital input 2
//     PlcTask Inputs/Axis6.biLimFwd <-> STM Status/Status/Digital input 1
//   Motion/Motion Instance <-> Device 1 (EtherCAT)/Term 14 (EK1200)/Term 24 (EL2004)
//     PlcTask Outputs/GVL_ver.AXIS{1..4}_Brake_q_disabled <-> Channel {1..4}/Output  (4 links)
//   Motion/Motion Instance <-> Device 1 (EtherCAT)/Term 14 (EK1200)/Term 25 (EL2004)
//     PlcTask Outputs/GVL_ver.AXIS5_Brake_q_disabled <-> Channel 1/Output
//     PlcTask Outputs/GVL_ver.AXIS6_Brake_q_disabled <-> Channel 2/Output
//   Motion/Motion Instance <-> Device 1 (EtherCAT)/Term 27 (EK1100)/Term 30 (EL7047)
//     PlcTask Inputs/Axis7.biLimBwd <-> STM Status/Status/Digital input 2
//     PlcTask Inputs/Axis7.biLimFwd <-> STM Status/Status/Digital input 1
//   Motion/Motion Instance <-> Device 1 (EtherCAT)/Term 27 (EK1100)/Term 31 (EL7047)
//     PlcTask Inputs/Axis8.biLimBwd <-> STM Status/Status/Digital input 2
//     PlcTask Inputs/Axis8.biLimFwd <-> STM Status/Status/Digital input 1
//   Motion/Motion Instance <-> Device 1 (EtherCAT)/Term 27 (EK1100)/Term 32 (EL7047)
//     PlcTask Inputs/Axis9.biLimBwd <-> STM Status/Status/Digital input 2
//     PlcTask Inputs/Axis9.biLimFwd <-> STM Status/Status/Digital input 1
//   Motion/Motion Instance <-> Device 1 (EtherCAT)/Term 27 (EK1100)/Term 46 (EL2004)
//     PlcTask Outputs/Axis1.boBrake <-> Channel 1/Output
//     PlcTask Outputs/MAIN.boBrake <-> Channel 2/Output
//   Motion/Motion Instance <-> NC-Task 1 SAF/Axes/Axis 1
//     PlcTask Inputs/Axis1.Axis.NcToPlc <-> Outputs/ToPlc
//     PlcTask Outputs/Axis1.Axis.PlcToNc <-> Inputs/FromPlc
//   Motion/Motion Instance <-> NC-Task 1 SAF/Axes/Axis 10
//     PlcTask Inputs/Axis10.Axis.NcToPlc <-> Outputs/ToPlc
//     PlcTask Outputs/Axis10.Axis.PlcToNc <-> Inputs/FromPlc
//   Motion/Motion Instance <-> NC-Task 1 SAF/Axes/Axis 2
//     PlcTask Inputs/Axis2.Axis.NcToPlc <-> Outputs/ToPlc
//     PlcTask Outputs/Axis2.Axis.PlcToNc <-> Inputs/FromPlc
//   Motion/Motion Instance <-> NC-Task 1 SAF/Axes/Axis 3
//     PlcTask Inputs/Axis3.Axis.NcToPlc <-> Outputs/ToPlc
//     PlcTask Outputs/Axis3.Axis.PlcToNc <-> Inputs/FromPlc
//   Motion/Motion Instance <-> NC-Task 1 SAF/Axes/Axis 4
//     PlcTask Inputs/Axis4.Axis.NcToPlc <-> Outputs/ToPlc
//     PlcTask Outputs/Axis4.Axis.PlcToNc <-> Inputs/FromPlc
//   Motion/Motion Instance <-> NC-Task 1 SAF/Axes/Axis 5
//     PlcTask Inputs/Axis5.Axis.NcToPlc <-> Outputs/ToPlc
//     PlcTask Outputs/Axis5.Axis.PlcToNc <-> Inputs/FromPlc
//   Motion/Motion Instance <-> NC-Task 1 SAF/Axes/Axis 6
//     PlcTask Inputs/Axis6.Axis.NcToPlc <-> Outputs/ToPlc
//     PlcTask Outputs/Axis6.Axis.PlcToNc <-> Inputs/FromPlc
//   Motion/Motion Instance <-> NC-Task 1 SAF/Axes/Axis 7
//     PlcTask Inputs/Axis7.Axis.NcToPlc <-> Outputs/ToPlc
//     PlcTask Outputs/Axis7.Axis.PlcToNc <-> Inputs/FromPlc
//   Motion/Motion Instance <-> NC-Task 1 SAF/Axes/Axis 8
//     PlcTask Inputs/Axis8.Axis.NcToPlc <-> Outputs/ToPlc
//     PlcTask Outputs/Axis8.Axis.PlcToNc <-> Inputs/FromPlc
//   Motion/Motion Instance <-> NC-Task 1 SAF/Axes/Axis 9
//     PlcTask Inputs/Axis9.Axis.NcToPlc <-> Outputs/ToPlc
//     PlcTask Outputs/Axis9.Axis.PlcToNc <-> Inputs/FromPlc

CONFIGURATION Motion
    RESOURCE PLC ON TwinCAT3
        TASK PlcTask(INTERVAL := T#10ms, PRIORITY := 20);
        PROGRAM MAIN WITH PlcTask : MAIN;
    END_RESOURCE
END_CONFIGURATION

// ---- GVLs/GVL_ver.TcGVL
{attribute 'qualified_only'}
VAR_GLOBAL
	Brake_i_disable AT %I* :BOOL;
	AXIS1_Brake_q_disabled AT %Q* :BOOL;
	AXIS2_Brake_q_disabled AT %Q* :BOOL;
	AXIS3_Brake_q_disabled AT %Q* :BOOL;
	AXIS4_Brake_q_disabled AT %Q* :BOOL;
	AXIS5_Brake_q_disabled AT %Q* :BOOL;
	AXIS6_Brake_q_disabled AT %Q* :BOOL;
	Axis4_ActPos AT %Q* :REAL;
	Axis4_ActVelo AT %Q* :REAL;
END_VAR

// ---- POUs/MAIN.TcPOU
PROGRAM MAIN
VAR
	fbPower: MC_POWER;
	biLimFwd AT %I*: BOOL;
	biLimBwd AT %I*: BOOL;
	boBrake AT %Q*:BOOL;
	bEnable: BOOL := TRUE;
	bHalt AT %Q*: BOOL ;
END_VAR


LadderLogic();

Axis1();
Axis2();
Axis3();
Axis4();
Axis5();
Axis6();

Axis7();
Axis8();
Axis9();
Axis10();

END_PROGRAM

// ---- POUs/LadderLogic.TcPOU
PROGRAM LadderLogic
VAR
	MC_Halt_0: MC_Halt;
END_VAR

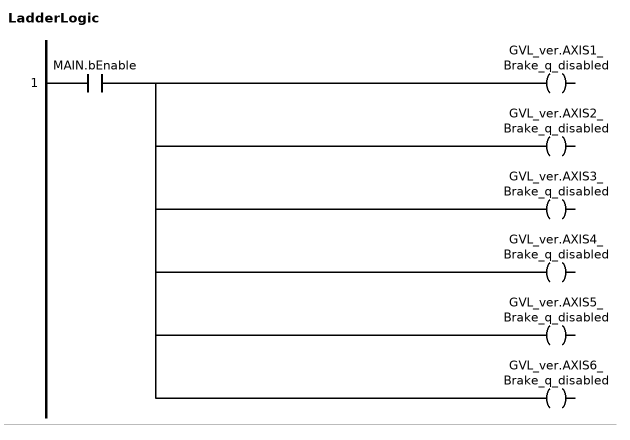
// NETWORK 1
GVL_ver.AXIS1_Brake_q_disabled := MAIN.bEnable;
GVL_ver.AXIS2_Brake_q_disabled := MAIN.bEnable;
GVL_ver.AXIS3_Brake_q_disabled := MAIN.bEnable;
GVL_ver.AXIS4_Brake_q_disabled := MAIN.bEnable;
GVL_ver.AXIS5_Brake_q_disabled := MAIN.bEnable;
GVL_ver.AXIS6_Brake_q_disabled := MAIN.bEnable;

END_PROGRAM

// ---- POUs/Axis2.TcPOU
PROGRAM Axis2
VAR
	fbPower: MC_POWER;
	Axis: AXIS_REF;
	biLimFwd AT %I*: BOOL;
	biLimBwd AT %I*: BOOL;
	boBrake AT %Q*:BOOL;
	bEnable: BOOL := TRUE;
	rPosition AT %Q*:REAL;
	rVelocity AT %Q*:REAL;
	roPosition AT %Q*:REAL;
	fbReadActialPosition: MC_ReadActualPosition;
	fbHalt: MC_Halt;
	boHalt AT%Q*:BOOL;
	fbMoveAbsolute: MC_MoveAbsolute;
	boMoveAbsolute AT%Q*:BOOL;
	fbReadActualVelocity: MC_ReadActualVelocity;
END_VAR

fbPower(Axis:=Axis,
	Enable:=bEnable,
	Enable_Positive:=biLimFwd,
	Enable_Negative:=biLimBwd);
boBrake:=bEnable;
fbReadActialPosition(
	Axis:=Axis , 
	Enable:=TRUE , 
	Valid=> , 
	Busy=> , 
	Error=> , 
	ErrorID=> , 
	Position=>rPosition );
fbHalt(
	Axis:=Axis , 
	Execute:=boHalt , 
	Deceleration:= , 
	Jerk:= , 
	BufferMode:= , 
	Options:= , 
	Done=>, 
	Busy=> , 
	Active=> , 
	CommandAborted=> , 
	Error=> , 
	ErrorID=> );
fbMoveAbsolute(
	Axis:=Axis , 
	Execute:=boMoveAbsolute , 
	Position:=roPosition , 
	Velocity:=0.1 , 
	Acceleration:= , 
	Deceleration:= , 
	Jerk:= , 
	BufferMode:= , 
	Options:= , 
	Done=> , 
	Busy=> , 
	Active=> , 
	CommandAborted=> , 
	Error=> , 
	ErrorID=> );
fbReadActualVelocity(
	Axis:=Axis , 
	Enable:=TRUE , 
	Valid=> , 
	Busy=> , 
	Error=> , 
	ErrorID=> , 
	ActualVelocity=>rVelocity );

END_PROGRAM

// ---- POUs/Axis4.TcPOU
PROGRAM Axis4
VAR
	fbPower: MC_POWER;
	Axis: AXIS_REF;
	biLimFwd AT %I*: BOOL;
	biLimBwd AT %I*: BOOL;
	boBrake AT %Q*:BOOL;
	bEnable: BOOL := TRUE;
	rPosition AT %Q*:REAL;
	rVelocity AT %Q*:REAL;
	roPosition AT %Q*:REAL;
	fbReadActialPosition: MC_ReadActualPosition;
	fbHalt: MC_Halt;
	boHalt AT%Q*:BOOL;
	fbMoveAbsolute: MC_MoveAbsolute;
	boMoveAbsolute AT%Q*:BOOL;
	fbReadActualVelocity: MC_ReadActualVelocity;
END_VAR

fbPower(Axis:=Axis,
	Enable:=bEnable,
	Enable_Positive:=biLimFwd,
	Enable_Negative:=biLimBwd);
boBrake:=bEnable;
fbReadActialPosition(
	Axis:=Axis , 
	Enable:=TRUE , 
	Valid=> , 
	Busy=> , 
	Error=> , 
	ErrorID=> , 
	Position=>rPosition );
fbHalt(
	Axis:=Axis , 
	Execute:=boHalt , 
	Deceleration:= , 
	Jerk:= , 
	BufferMode:= , 
	Options:= , 
	Done=>, 
	Busy=> , 
	Active=> , 
	CommandAborted=> , 
	Error=> , 
	ErrorID=> );
fbMoveAbsolute(
	Axis:=Axis , 
	Execute:=boMoveAbsolute , 
	Position:=roPosition , 
	Velocity:=0.1 , 
	Acceleration:= , 
	Deceleration:= , 
	Jerk:= , 
	BufferMode:= , 
	Options:= , 
	Done=> , 
	Busy=> , 
	Active=> , 
	CommandAborted=> , 
	Error=> , 
	ErrorID=> );
fbReadActualVelocity(
	Axis:=Axis , 
	Enable:=TRUE , 
	Valid=> , 
	Busy=> , 
	Error=> , 
	ErrorID=> , 
	ActualVelocity=>rVelocity );

END_PROGRAM

// ---- POUs/Axis8.TcPOU
PROGRAM Axis8
VAR
	fbPower: MC_POWER;
	Axis: AXIS_REF;
	biLimFwd AT %I*: BOOL;
	biLimBwd AT %I*: BOOL;
	boBrake AT %Q*:BOOL;
	bEnable: BOOL := TRUE;
	rPosition AT %Q*:REAL;
	rVelocity AT %Q*:REAL;
	roPosition AT %Q*:REAL;
	fbReadActialPosition: MC_ReadActualPosition;
	fbHalt: MC_Halt;
	boHalt AT%Q*:BOOL;
	fbMoveAbsolute: MC_MoveAbsolute;
	boMoveAbsolute AT%Q*:BOOL;
	fbReadActualVelocity: MC_ReadActualVelocity;
END_VAR

fbPower(Axis:=Axis,
	Enable:=bEnable,
	Enable_Positive:=biLimFwd,
	Enable_Negative:=biLimBwd);
boBrake:=bEnable;
fbReadActialPosition(
	Axis:=Axis , 
	Enable:=TRUE , 
	Valid=> , 
	Busy=> , 
	Error=> , 
	ErrorID=> , 
	Position=>rPosition );
fbHalt(
	Axis:=Axis , 
	Execute:=boHalt , 
	Deceleration:= , 
	Jerk:= , 
	BufferMode:= , 
	Options:= , 
	Done=>, 
	Busy=> , 
	Active=> , 
	CommandAborted=> , 
	Error=> , 
	ErrorID=> );
fbMoveAbsolute(
	Axis:=Axis , 
	Execute:=boMoveAbsolute , 
	Position:=roPosition , 
	Velocity:=0.1 , 
	Acceleration:= , 
	Deceleration:= , 
	Jerk:= , 
	BufferMode:= , 
	Options:= , 
	Done=> , 
	Busy=> , 
	Active=> , 
	CommandAborted=> , 
	Error=> , 
	ErrorID=> );
fbReadActualVelocity(
	Axis:=Axis , 
	Enable:=TRUE , 
	Valid=> , 
	Busy=> , 
	Error=> , 
	ErrorID=> , 
	ActualVelocity=>rVelocity );

END_PROGRAM

// ---- POUs/Axis10.TcPOU
PROGRAM Axis10
VAR
	fbPower: MC_POWER;
	Axis: AXIS_REF;
	biLimFwd AT %I*: BOOL:=TRUE;
	biLimBwd AT %I*: BOOL:=TRUE;
	boBrake AT %Q*:BOOL;
	bEnable: BOOL := TRUE;
	rPosition AT %Q*:REAL;
	rVelocity AT %Q*:REAL;
	roPosition AT %Q*:REAL;
	fbReadActialPosition: MC_ReadActualPosition;
	fbHalt: MC_Halt;
	boHalt AT%Q*:BOOL;
	fbMoveAbsolute: MC_MoveAbsolute;
	boMoveAbsolute AT%Q*:BOOL;
	fbReadActualVelocity: MC_ReadActualVelocity;
	Enable_Nagative: STRING(INT#4);
	Enable: BOOL;
	Enable_Positive: BOOL;
	Enable_Negative: BOOL;
END_VAR

fbPower(Axis:=Axis,
	Enable:=bEnable,
	Enable_Positive:=TRUE,
	Enable_Negative:=TRUE);
boBrake:=bEnable;
fbReadActialPosition(
	Axis:=Axis , 
	Enable:=TRUE , 
	Valid=> , 
	Busy=> , 
	Error=> , 
	ErrorID=> , 
	Position=>rPosition );
fbHalt(
	Axis:=Axis , 
	Execute:=boHalt , 
	Deceleration:= , 
	Jerk:= , 
	BufferMode:= , 
	Options:= , 
	Done=>, 
	Busy=> , 
	Active=> , 
	CommandAborted=> , 
	Error=> , 
	ErrorID=> );
fbMoveAbsolute(
	Axis:=Axis , 
	Execute:=boMoveAbsolute , 
	Position:=roPosition , 
	Velocity:=0.1 , 
	Acceleration:= , 
	Deceleration:= , 
	Jerk:= , 
	BufferMode:= , 
	Options:= , 
	Done=> , 
	Busy=> , 
	Active=> , 
	CommandAborted=> , 
	Error=> , 
	ErrorID=> );
fbReadActualVelocity(
	Axis:=Axis , 
	Enable:=TRUE , 
	Valid=> , 
	Busy=> , 
	Error=> , 
	ErrorID=> , 
	ActualVelocity=>rVelocity );

END_PROGRAM

// ---- POUs/GCC1.TcPOU
PROGRAM GCC1
VAR
	rfbAdsRead: ADSREAD;
	sNetId: T_AmsNetID:='192.168.0.3';
	sPort: T_AmsPort:=851;
	bRead:BOOL:=TRUE;
	rPress: REAL;
	bPress: BOOL;
END_VAR

rfbAdsRead(
	NETID:= sNetID , 
	PORT:= sPort, 
	IDXGRP:= 16#4040, 
	IDXOFFS:= 971100, 
	LEN:= SIZEOF(bPress),
	DESTADDR:= ADR(bPress) , 
	READ:= bRead);

END_PROGRAM

// ---- VISUs/StandMotors.TcVIS
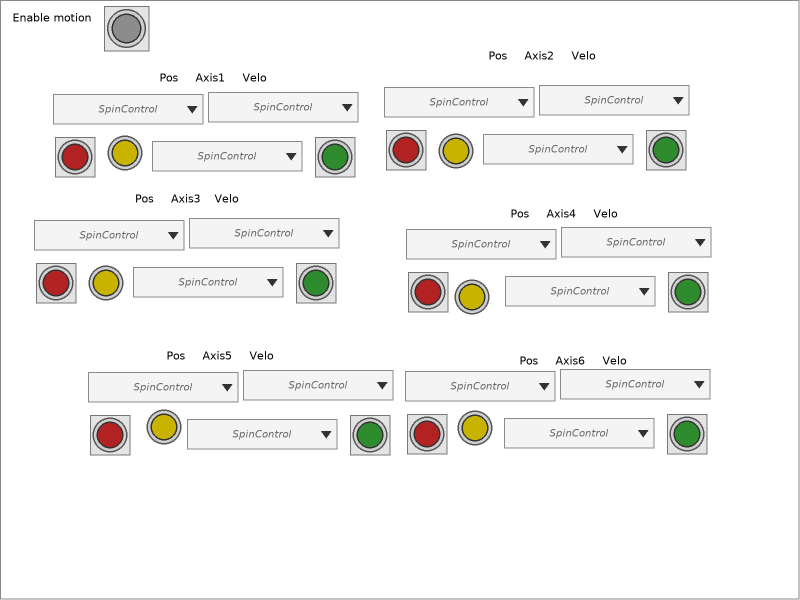
VISUALIZATION StandMotors  // 800x600
    PushSwitch (104,2 45x53), variable: MAIN.bEnable, behaviour: TOGGLE, style: Switch-PushSwitch-Gray
    Lamp1 (105,133 40x40), variable: GVL_ver.AXIS1_Brake_q_disabled, style: Lamp-Lamp1-Yellow
    Label (8,3 88x30), "Enable motion"
    Lamp1 (436,131 40x40), variable: GVL_ver.AXIS2_Brake_q_disabled, style: Lamp-Lamp1-Yellow
    Lamp1 (86,263 40x40), variable: GVL_ver.AXIS3_Brake_q_disabled, style: Lamp-Lamp1-Yellow
    Lamp1 (452,277 40x40), variable: GVL_ver.AXIS4_Brake_q_disabled, style: Lamp-Lamp1-Yellow
    Lamp1 (144,407 40x40), variable: GVL_ver.AXIS5_Brake_q_disabled, style: Lamp-Lamp1-Yellow
    Lamp1 (455,408 40x40), variable: GVL_ver.AXIS6_Brake_q_disabled, style: Lamp-Lamp1-Yellow
    SpinControl (406,229 150x30), variable: Axis4.rPosition
    PushSwitch (408,272 40x40), variable: Axis4.boHalt, behaviour: TOGGLE, style: Switch-PushSwitch-Red
    PushSwitch (668,272 40x40), variable: Axis4.boMoveAbsolute, behaviour: TOGGLE, style: Switch-PushSwitch-Green
    SpinControl (505,276 150x30), variable: Axis4.roPosition
        p1653691745: 0.05
    SpinControl (561,227 150x30), variable: Axis4.rVelocity
        p1653691745: 0.05
    Label (489,199 150x30), "Pos Axis4 Velo"
    Label (498,346 150x30), "Pos Axis6 Velo"
    Label (145,341 150x30), "Pos Axis5 Velo"
    PushSwitch (36,263 40x40), variable: Axis3.boHalt, behaviour: TOGGLE, style: Switch-PushSwitch-Red
    SpinControl (34,220 150x30), variable: Axis3.rPosition
    PushSwitch (296,263 40x40), variable: Axis3.boMoveAbsolute, behaviour: TOGGLE, style: Switch-PushSwitch-Green
    SpinControl (133,267 150x30), variable: Axis3.roPosition
        p1653691745: 0.05
    SpinControl (189,218 150x30), variable: Axis3.rVelocity
        p1653691745: 0.05
    PushSwitch (386,130 40x40), variable: Axis2.boHalt, behaviour: TOGGLE, style: Switch-PushSwitch-Red
    SpinControl (384,87 150x30), variable: Axis2.rPosition
    PushSwitch (646,130 40x40), variable: Axis2.boMoveAbsolute, behaviour: TOGGLE, style: Switch-PushSwitch-Green
    SpinControl (483,134 150x30), variable: Axis2.roPosition
        p1653691745: 0.05
    SpinControl (539,85 150x30), variable: Axis2.rVelocity
        p1653691745: 0.05
    PushSwitch (55,137 40x40), variable: Axis1.boHalt, behaviour: TOGGLE, style: Switch-PushSwitch-Red
    SpinControl (53,94 150x30), variable: Axis1.rPosition
    PushSwitch (315,137 40x40), variable: Axis1.boMoveAbsolute, behaviour: TOGGLE, style: Switch-PushSwitch-Green
    SpinControl (152,141 150x30), variable: Axis1.roPosition
        p1653691745: 0.05
    SpinControl (208,92 150x30), variable: Axis1.rVelocity
        p1653691745: 0.05
    PushSwitch (407,414 40x40), variable: Axis6.boHalt, behaviour: TOGGLE, style: Switch-PushSwitch-Red
    SpinControl (405,371 150x30), variable: Axis6.rPosition
    PushSwitch (667,414 40x40), variable: Axis6.boMoveAbsolute, behaviour: TOGGLE, style: Switch-PushSwitch-Green
    SpinControl (504,418 150x30), variable: Axis6.roPosition
        p1653691745: 0.05
    SpinControl (560,369 150x30), variable: Axis6.rVelocity
        p1653691745: 0.05
    PushSwitch (90,415 40x40), variable: Axis5.boHalt, behaviour: TOGGLE, style: Switch-PushSwitch-Red
    SpinControl (88,372 150x30), variable: Axis5.rPosition
    PushSwitch (350,415 40x40), variable: Axis5.boMoveAbsolute, behaviour: TOGGLE, style: Switch-PushSwitch-Green
    SpinControl (187,419 150x30), variable: Axis5.roPosition
        p1653691745: 0.05
    SpinControl (243,370 150x30), variable: Axis5.rVelocity
        p1653691745: 0.05
    Label (112,184 150x30), "Pos Axis3 Velo"
    Label (467,41 150x30), "Pos Axis2 Velo"
    Label (138,63 150x30), "Pos Axis1 Velo"
END_VISUALIZATION

// ---- VISUs/ManiMotors.TcVIS
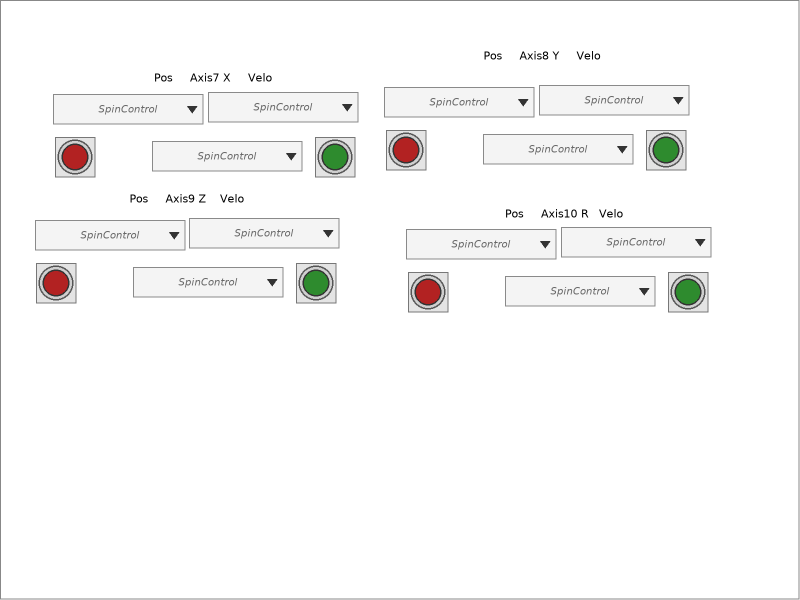
VISUALIZATION ManiMotors  // 800x600
    SpinControl (406,229 150x30), variable: Axis10.rPosition
    PushSwitch (408,272 40x40), variable: Axis10.boHalt, behaviour: TOGGLE, style: Switch-PushSwitch-Red
    PushSwitch (668,272 40x40), variable: Axis10.boMoveAbsolute, behaviour: TOGGLE, style: Switch-PushSwitch-Green
    SpinControl (505,276 150x30), variable: Axis10.roPosition
    SpinControl (561,227 150x30), variable: Axis10.rVelocity
    Label (489,199 150x30), "Pos Axis10 R Velo"
    PushSwitch (36,263 40x40), variable: Axis9.boHalt, behaviour: TOGGLE, style: Switch-PushSwitch-Red
    SpinControl (35,220 150x30), variable: Axis9.rPosition
    PushSwitch (296,263 40x40), variable: Axis9.boMoveAbsolute, behaviour: TOGGLE, style: Switch-PushSwitch-Green
    SpinControl (133,267 150x30), variable: Axis9.roPosition
        p1653691745: 0.05
    SpinControl (189,218 150x30), variable: Axis9.rVelocity
    PushSwitch (386,130 40x40), variable: Axis8.boHalt, behaviour: TOGGLE, style: Switch-PushSwitch-Red
    SpinControl (384,87 150x30), variable: Axis8.rPosition
    PushSwitch (646,130 40x40), variable: Axis8.boMoveAbsolute, behaviour: TOGGLE, style: Switch-PushSwitch-Green
    SpinControl (483,134 150x30), variable: Axis8.roPosition
        p1653691745: 0.05
    SpinControl (539,85 150x30), variable: Axis8.rVelocity
    PushSwitch (55,137 40x40), variable: Axis7.boHalt, behaviour: TOGGLE, style: Switch-PushSwitch-Red
    SpinControl (53,94 150x30), variable: Axis7.rPosition
    PushSwitch (315,137 40x40), variable: Axis7.boMoveAbsolute, behaviour: TOGGLE, style: Switch-PushSwitch-Green
    SpinControl (152,141 150x30), variable: Axis7.roPosition
        p1653691745: 0.05
    SpinControl (208,92 150x30), variable: Axis7.rVelocity
    Label (112,184 150x30), "Pos Axis9 Z Velo"
    Label (467,41 150x30), "Pos Axis8 Y Velo"
    Label (138,63 150x30), "Pos Axis7 X Velo"
END_VISUALIZATION
